TEXTLIST TL_Params_BOOL
  1 = 'UseCooling' | en: 'a' | de: 'a'
  2 = 'ExtruderCompEna'
  3 = 'TuneCooling'
  4 = 'Tune_IdleLoad'
  5 = 'Autotune'
  6 = 'Enable'
  7 = 'Update'
  8 = 'EnaExtruderBlock'
  9 = 'NoFanWhileTrackDown'
  10 = 'Ena_TuneIdleLoad'
  11 = 'LooptestUpdate'
  12 = 'EnableErrorHeating'
  13 = 'ReadBack'
  14 = 'TuneExtruderComp'
  15 = 'TuneHeaterLoad'
  16 = 'OpenloopHeating'
  17 = 'fc_Enable'
  18 = 'HibernateI_Cool'
  19 = 'hibernateI_Heat'
  20 = 'bSavingParams'
  21 = 'bLoadParams'
  22 = '*** not Used ***'
  23 = '*** not Used ***'
  24 = '*** not Used ***'
  25 = '*** not Used ***'
  26 = '*** not Used ***'
  27 = '*** not Used ***'
  28 = '*** not Used ***'
  29 = '*** not Used ***'
  30 = '*** not Used ***'
  31 = '*** not Used ***'
  32 = '*** not Used ***'
  33 = '*** not Used ***'
  34 = '*** not Used ***'
  35 = '*** not Used ***'
  36 = '*** not Used ***'
  37 = '*** not Used ***'
  38 = '*** not Used ***'
  39 = '*** not Used ***'
  40 = '*** not Used ***'
   = ''
END_TEXTLIST

(* stored: Version 1.1.0.1, ProductVersion 3.1.4020.12
   TextList TL_Params_BOOL: Id {c863ecfe-bc02-4c16-a5a3-862fcdb22c95} *)
